// TIA Portal V18 export
DATA_BLOCK "AHUSetPoints"   // DB106
{ S7_Optimized_Access := 'FALSE' }
VERSION : 0.1
// stored: AutoNumber false, DBAccessibleFromOPCUA true, IsOnlyStoredInLoadMemory false, IsWriteProtectedInAS false
   VAR RETAIN
      SetPoints { S7_SetPoint := 'True'} : "UDT_AHUSetpoints";
   END_VAR
BEGIN
END_DATA_BLOCK
